// TwinCAT 3 PLC project _02_Decorator
// ProgramVersion: 3.1.4023.0
// libraries:
//   Tc2_Standard, * (Beckhoff Automation GmbH)
//   Tc2_System, * (Beckhoff Automation GmbH)
//   Tc2_Utilities, * (Beckhoff Automation GmbH)
//   Tc3_Module, * (Beckhoff Automation GmbH)
// project tree:
//   Decorator Pattern/ P_Decorator.TcPOU
//   Decorator Pattern/StringBuilder/ StringBuilder.TcPOU
//   / MAIN.TcPOU, PlcTask.TcTTO
// real-time tasks:
//   TASK PlcTask: cycle T#10ms, priority 20, ADS port 350
// motion (NC):
//   TASK NC-Task 1 SAF: cycle T#2ms, priority 4, ADS port 501
//   TASK NC-Task 1 SVB: cycle T#10ms, priority 8, ADS port 511
//   AXIS FacadeAxis (id 1)
// variable links:
//   14_Facade Instance <-> NC-Task 1 SAF/Axes/FacadeAxis
//     PlcTask Inputs/MAIN.axisControl._axis.NcToPlc <-> Outputs/ToPlc
//     PlcTask Outputs/MAIN.axisControl._axis.PlcToNc <-> Inputs/FromPlc

CONFIGURATION _02_Decorator
    RESOURCE PLC ON TwinCAT3
        TASK PlcTask(INTERVAL := T#10ms, PRIORITY := 20);
        PROGRAM MAIN WITH PlcTask : MAIN;
    END_RESOURCE
END_CONFIGURATION

// ---- MAIN.TcPOU
PROGRAM MAIN
VAR
END_VAR

(* 
	GOF 		Attach additional responsibilities to an object dynamically. Decorators
				provide a flexible alternative to subclassing for extending functionality.   
*)
P_Decorator();

END_PROGRAM

// ---- Decorator Pattern/P_Decorator.TcPOU
PROGRAM P_Decorator
VAR
	ErrorString				: STRING;
	stringBuilder			: StringBuilder;
	ErrorNumber				: INT := 1;
	ErrorMessage			: STRING := 'This is my error message';
END_VAR

ErrorString := stringBuilder
					.Clear()
					.Append('Error number: ')
					.Append(INT_TO_STRING(ErrorNumber))
					.Append('. Message: ')
					.Append(ErrorMessage)
					.Append('.')
					.ToString();

END_PROGRAM

// ---- Decorator Pattern/StringBuilder/StringBuilder.TcPOU
// Copyright (c) 2020 Dustin Hullett, Inxton team, MTS spol. s r.o. and contributors
(*~
<docu>
	<summary>
			Allows to concat strings using fluent interface. It's similar to C# StringBuilder class
			Usage as follows :
			<code>
				ErrorString := _stringBuilder
					.Clear()
					.Append('Error number: ')
					.Append(INT_TO_STRING(ErrorNumber))
					.Append('. Message: ')
					.Append(ErrorMessage)
					.Append('.')
					.ToString();
			</code>
			
			Inspired by Gerhard Barteling blogpost at https://www.plccoder.com/fluent-code/
	</summary>				
</docu>	
~*)	
FUNCTION_BLOCK StringBuilder
VAR
	{attribute 'hide'}
    _workString						: T_MAXSTRING;
END_VAR

(*
	Thanks to https://github.com/bengeisler/TcLog
*)

METHOD PROTECTED AnyToString : STRING(255)
VAR_INPUT
	Data:	ANY;
END_VAR
VAR
	pAnyBOOL		: POINTER TO BOOL; 
	pAnyBYTE		: POINTER TO BYTE; 
	pAnyWORD		: POINTER TO WORD; 
	pAnyDWORD		: POINTER TO DWORD;
	pAnyLWORD		: POINTER TO LWORD;
	pAnySINT		: POINTER TO SINT; 
	pAnyUSINT		: POINTER TO USINT;
	pAnyINT			: POINTER TO INT;  
	pAnyUINT		: POINTER TO UINT; 
	pAnyDINT		: POINTER TO DINT; 
	pAnyUDINT		: POINTER TO UDINT;
	pAnyLINT		: POINTER TO LINT; 
	pAnyULINT		: POINTER TO ULINT;
	pAnyLTIME		: POINTER TO LTIME;	
	pAnyReal 		: POINTER TO REAL;
	pAnyLReal		: POINTER TO LREAL;	
	pAnyDateAndTime : POINTER TO DATE_AND_TIME;
	pAnyDate		: POINTER TO DATE;
	pAnyTime		: POINTER TO TIME;
	pAnyWString		: POINTER TO WSTRING;
	pAnyTOD			: POINTER TO TOD;
	pAnyString		: POINTER TO STRING;	
	sString			: T_MAXSTRING;
	wWString		: WSTRING;
END_VAR
IF Data.TypeClass = __SYSTEM.TYPE_CLASS.TYPE_REAL THEN
	pAnyReal := Data.pValue;
	AnyToString := REAL_TO_STRING(pAnyReal^);
	
ELSIF Data.TypeClass = __SYSTEM.TYPE_CLASS.TYPE_LREAL THEN
	pAnyLReal := Data.pValue;
	AnyToString := LREAL_TO_STRING(pAnyLReal^);
	
ELSIF Data.TypeClass = __SYSTEM.TYPE_CLASS.TYPE_DATEANDTIME THEN
	pAnyDateAndTime := Data.pValue;
	AnyToString := DT_TO_STRING(pAnyDateAndTime^);	
	
ELSIF Data.TypeClass = __SYSTEM.TYPE_CLASS.TYPE_DATE THEN
	pAnyDate := Data.pValue;
	AnyToString := DATE_TO_STRING(pAnyDate^);
	
ELSIF Data.TypeClass = __SYSTEM.TYPE_CLASS.TYPE_TIME THEN
	pAnyTime := Data.pValue;
	AnyToString := TIME_TO_STRING(pAnyTime^);
	
ELSIF Data.TypeClass = __SYSTEM.TYPE_CLASS.TYPE_STRING THEN
	pAnyString := Data.pValue;
	AnyToString := pAnyString^;
	
ELSIF Data.TypeClass = __SYSTEM.TYPE_CLASS.TYPE_WSTRING THEN
	pAnyWString := Data.pValue;
	wWString := pAnyWString^;
	WSTRING_TO_STRING2(ADR(sString), ADR(wWstring), SIZEOF(wWString));
	AnyToString := sString;
	
ELSIF Data.TypeClass = __SYSTEM.TYPE_CLASS.TYPE_TIMEOFDAY THEN
	pAnyTOD := Data.pValue;
	AnyToString := TOD_TO_STRING(pAnyTOD^);
ELSIF Data.TypeClass = __SYSTEM.TYPE_CLASS.TYPE_BOOL THEN 	
	pAnyBOOL := Data.pValue;
	AnyToString := BOOL_TO_STRING(pAnyBool^);
ELSIF Data.TypeClass = __SYSTEM.TYPE_CLASS.TYPE_BYTE THEN
	pAnyBYTE := Data.pValue;
	AnyToString := BYTE_TO_STRING(pAnyBYTE^);	
ELSIF Data.TypeClass = __SYSTEM.TYPE_CLASS.TYPE_WORD THEN
	pAnyWORD := Data.pValue;
	AnyToString := WORD_TO_STRING(pAnyWORD^);	
ELSIF Data.TypeClass = __SYSTEM.TYPE_CLASS.TYPE_DWORD THEN
	pAnyDWORD := Data.pValue;	
	AnyToString := DWORD_TO_STRING(pAnyDWORD^);
ELSIF Data.TypeClass = __SYSTEM.TYPE_CLASS.TYPE_LWORD THEN
	pAnyLWORD := Data.pValue;	
	AnyToString := LWORD_TO_STRING(pAnyLWORD^);
ELSIF Data.TypeClass = __SYSTEM.TYPE_CLASS.TYPE_SINT THEN
	pAnySINT := Data.pValue;	
	AnyToString := SINT_TO_STRING(pAnySINT^);					
ELSIF Data.TypeClass = __SYSTEM.TYPE_CLASS.TYPE_USINT THEN
	pAnyUSINT := Data.pValue;	
	AnyToString := USINT_TO_STRING(pAnyUSINT^);	
ELSIF Data.TypeClass = __SYSTEM.TYPE_CLASS.TYPE_INT THEN
	pAnyINT := Data.pValue;	
	AnyToString := INT_TO_STRING(pAnyINT^);	
ELSIF Data.TypeClass = __SYSTEM.TYPE_CLASS.TYPE_UINT THEN
	pAnyUINT := Data.pValue;	
	AnyToString := UINT_TO_STRING(pAnyUINT^);	
ELSIF Data.TypeClass = __SYSTEM.TYPE_CLASS.TYPE_DINT THEN
	pAnyDINT := Data.pValue;	
	AnyToString := DINT_TO_STRING(pAnyDINT^);	
ELSIF Data.TypeClass = __SYSTEM.TYPE_CLASS.TYPE_UDINT THEN
	pAnyUDINT := Data.pValue;	
	AnyToString := UDINT_TO_STRING(pAnyUDINT^);	
ELSIF Data.TypeClass = __SYSTEM.TYPE_CLASS.TYPE_LINT THEN
	pAnyLINT := Data.pValue;	
	AnyToString := LINT_TO_STRING(pAnyLINT^);	
ELSIF Data.TypeClass = __SYSTEM.TYPE_CLASS.TYPE_ULINT THEN
	pAnyULINT := Data.pValue;	
	AnyToString := ULINT_TO_STRING(pAnyULINT^);	
ELSIF Data.TypeClass = __SYSTEM.TYPE_CLASS.TYPE_LTIME THEN
	pAnyLTIME := Data.pValue;	
	AnyToString := LTIME_TO_STRING(pAnyLTIME^);		
ELSE	
	AnyToString := ANY_TO_STRING(Data.pValue^);
END_IF
END_METHOD

METHOD Append : REFERENCE TO StringBuilder
VAR_INPUT
    Text :STRING(255); 
END_VAR
_workString := Concat(_workString,text);
Append REF= THIS^;
END_METHOD

METHOD INTERNAL AppendAny : REFERENCE TO StringBuilder
VAR_INPUT
	Data : ANY;
END_VAR
_workString := Concat(_workString,AnyToString(Data));
AppendAny REF= THIS^;
END_METHOD

METHOD Clear : REFERENCE TO StringBuilder
_workString := '';
Clear REF= THIS^;
END_METHOD

METHOD ToString : T_MAXSTRING
ToString := _workString;
END_METHOD

END_FUNCTION_BLOCK
